{attribute 'qualified_only'}
{attribute 'strict'}
{attribute 'to_string'}
TYPE E_TestStatus : (
		Init := 0,
		Running,
		DoneOk,
		DoneFailed
	);
END_TYPE

(* stored: Version 1.1.0.1
   DUT E_TestStatus: Id {ea72af65-669a-4172-8425-0b7ea0ae6c93} *)
